(* CODESYS project Manutec_r2.project

Project tree, tasks and I/O mapping:
  Manutec : CODESYS SoftMotion Win V3, 3S - Smart Software Solutions GmbH, order no. 309021, version 3.5.9.20
    application Application
      libraries: SysSocket, * (System)
      task Manu_PlanningTask (cyclic, interval t#1000ms, priority 2) calls Manutech_PlanningPrg, Server
      task Task (cyclic, interval t#20ms, priority 1) calls RoboterSteuerung, qSoll
      task VISU_TASK (cyclic, interval 100 ms, priority 31) calls VisuElems.Visu_Prg
      axis group Manutech: TRAFO.Kin_ArticulatedRobot_6DOF, axes DriveA1, DriveA2, DriveA3, DriveA4, DriveA5, DriveA6
      program Manutech_PlanningPrg [ST]
      program RoboterSteuerung [FBD]
      global variables GVL
      visualisation Visualization
      visualisation VIS_Arm2
      data type CLIENT_ACCEPT
      data type SOCKET_LINGER
      TCP/
        function TcpReceiveData [ST]
        function TcpSendData [ST]
        function TcpServerOpenSocket [ST]
        function TcpServerWaitForConnect [ST]
        function block Tcp_Server [ST]
      program Server [FBD]
      program qSoll [ST]
    SoftMotion General Axis Pool
      DriveA1 : SM_Drive_Virtual, 3S - Smart Software Solutions GmbH, order no. 1805, version 4.0.0.0
          settings: wDriveID = 0; fSWMaxAcceleration = 100; fSWMaxDeceleration = 100; fSWMaxJerk = 1000; fSWLimitPositive = 360; fSWLimitNegative = 0; fSWLimitDeceleration = 0.0; fSWErrorMaxDistance = 0.0
      DriveA2 : SM_Drive_Virtual, 3S - Smart Software Solutions GmbH, order no. 1805, version 4.0.0.0
          settings: fSWMaxAcceleration = 100; fSWMaxDeceleration = 100; fSWMaxJerk = 1000; fSWLimitPositive = 90; fSWLimitNegative = -90
      DriveA3 : SM_Drive_Virtual, 3S - Smart Software Solutions GmbH, order no. 1805, version 4.0.0.0
          settings: wDriveID = 2; fSWLimitPositive = 180; fSWLimitNegative = -180; bSWLimitEnable = TRUE
      DriveA4 : SM_Drive_Virtual, 3S - Smart Software Solutions GmbH, order no. 1805, version 4.0.0.0
          settings: wDriveID = 3
      DriveA5 : SM_Drive_Virtual, 3S - Smart Software Solutions GmbH, order no. 1805, version 4.0.0.0
          settings: wDriveID = 4
      DriveA6 : SM_Drive_Virtual, 3S - Smart Software Solutions GmbH, order no. 1805, version 4.0.0.0
          settings: wDriveID = 5
  text list GlobalTextList
*)

// Manutec/Application/CLIENT_ACCEPT
TYPE  CLIENT_ACCEPT :
STRUCT
	Socket:DINT;       (* Socket Id des Client  *)
	IPAddress:STRING(20);	(* IP Adresse des Client *)
END_STRUCT
END_TYPE

// Manutec/Application/SOCKET_LINGER
TYPE  SOCKET_LINGER :
STRUCT
	l_onoff:WORD;
	l_linger:WORD;
END_STRUCT
END_TYPE

// Manutec/Application/GVL
VAR_GLOBAL CONSTANT
	PI: REAL := 3.141592654;
END_VAR
VAR_GLOBAL
	AxisMove: BOOL;
	PtpMOVE : BOOL;
	MoveLin: BOOL;
	Ziel : SMC_POS_REF;
	SOCKET_INVALID : DINT := -1;
	Port:INT:=2000;
	qAct:ARRAY[1..8] OF REAL;;
END_VAR

// Manutec/Application/Manutech_PlanningPrg
PROGRAM Manutech_PlanningPrg

;

END_PROGRAM

// Manutec/Application/Server
PROGRAM  Server
VAR
		Server: TCP_Server;
END_VAR

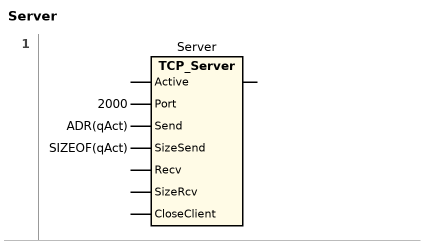
// NETWORK 1
Server(Port := 2000, Send := ADR(qAct), SizeSend := SIZEOF(qAct)); // TCP_Server

END_PROGRAM

// Manutec/Application/TCP/Tcp_Server
FUNCTION_BLOCK Tcp_Server
VAR_INPUT
	Active: BOOL;
	Port : INT;							(* zum Datenaustausch verwendeter Port *)
	Send : DWORD;					(* Sende Daten *)
	SizeSend : DINT;
	Recv : DWORD;					(* Empfangs Daten *)
	SizeRcv : DINT;
	CloseClient: BOOL;							(*Client schließen*)
END_VAR
VAR_OUTPUT

END_VAR
VAR
	Socket : DINT := -1;						(* Socket Id (wird von FUN "TcpServerOpenSocket" erzeugt) *)
	Client : CLIENT_ACCEPT := (Socket := -1);


END_VAR

IF Active THEN		(* Wenn Server aktiv dann ... *)
	IF Socket = -1 THEN		(* Wenn noch kein Server Socket geöffnet, dann ... *)
		Socket := TcpServerOpenSocket(Port, 10, 1000); (* ... Server Socket öffnen *)
		END_IF
	IF  Client.Socket = -1 THEN		(* Wenn noch kein Client verbuden, dann...   *)
		Client := TcpServerWaitForConnect(Socket, 4);	(*... warten auf Verbindung*)
	END_IF
	IF  Client.Socket <> -1 THEN	(* Wenn ein Client verbuden, dann...   *)
		TcpSendData(Client.Socket, Send, SizeSend, 1);		(* ... Daten senden *)
		TcpReceiveData(Client.Socket, Recv, SizeRcv, 5);	(* Daten empfangen *)
	END_IF
	IF CloseClient THEN		(* Wenn Client geschlossen werden soll, dann... *)
		CloseClient := FALSE;		(* ... Schließbefehl wieder auf FALSE setzen   *)
		SysSockClose(hSocket:=Client.Socket);	(* Client Socket schließen  *)
		Client.Socket := -1;		(* Client Socket wieder auf Startwert setzen *)
	END_IF
END_IF

END_FUNCTION_BLOCK

// Manutec/Application/TCP/TcpServerOpenSocket
FUNCTION TcpServerOpenSocket :  DINT
(*	Open a TCP server socket.
	Return:	Main Socket Id
*)
VAR_INPUT
	iPort:INT;						(* Port number *)
	diMaxConnections:DINT;		(* Max possible client connections of the server *)
	diMaxDataSize:DINT;			(* Max size of data to transmitt; if size = 0 default values are used *)
END_VAR
VAR
	diSocket:DINT;
	pResult:UDINT;  //Funktion überprüfen
	sa:SOCKADDRESS;
	bOptNoDelay:BOOL;
	lOptLinger:SOCKET_LINGER;
	
END_VAR

diSocket:=SysSockCreate(SOCKET_AF_INET, SOCKET_STREAM, 0, pResult);
IF diSocket <> SOCKET_INVALID THEN
(*
	IF diMaxDataSize <> 0 THEN
		SysSockSetOption(diSocket, SOCKET_SOL, SOCKET_SO_SNDBUF, ADR(diMaxDataSize), SIZEOF(diMaxDataSize));
		SysSockSetOption(diSocket, SOCKET_SOL, SOCKET_SO_RCVBUF, ADR(diMaxDataSize), SIZEOF(diMaxDataSize));
	END_IF
	lOptLinger.l_onoff:=0;
	lOptLinger.l_linger:=0;
	SysSockSetOption(diSocket,	SOCKET_SOL, SOCKET_SO_LINGER, ADR(lOptLinger), SIZEOF(lOptLinger));
	bOptNoDelay:=TRUE;
	SysSockSetOption(diSocket,	SOCKET_IPPROTO_TCP, SOCKET_TCP_NODELAY, ADR(bOptNoDelay), SIZEOF(bOptNoDelay));
*)

	sa.sin_family:=SOCKET_AF_INET;
	sa.sin_addr.ulAddr:=SOCKET_INADDR_ANY;
	sa.sin_port:=SysSockHtons(iPort);
	pResult:=SysSockBind(diSocket, ADR(sa), SIZEOF(sa));
	IF pResult >0 THEN
		diSocket:=SOCKET_INVALID;
	ELSE
		pResult:=SysSockListen(diSocket, diMaxConnections);
		IF pResult >0 THEN
			diSocket:=SOCKET_INVALID;
		END_IF
	END_IF
END_IF
TcpServerOpenSocket:=diSocket;

END_FUNCTION

// Manutec/Application/TCP/TcpServerWaitForConnect
FUNCTION TcpServerWaitForConnect : CLIENT_ACCEPT
(*	Wait for a TCP client to connect.
	ATTENTION:  Function is blocking, until a client tries to connect!
	Return:	diSocket : Socket Id for connection session
				stIPAddress : IP-Address of connected client
*)
VAR_INPUT
	diServerSocket:DINT;
	diTimeout : DINT;	(* Timeout in seconds *)
END_VAR
VAR
	sa:SOCKADDRESS;
	ia:INADDR;
	diSize:DINT;
	presult : UDINT;    //funktion überprüfen
	fdRead: SOCKET_FD_SET;
	fdWrite:SOCKET_FD_SET;
	fdExcept:SOCKET_FD_SET;
	tvTimeout:SOCKET_TIMEVAL;
END_VAR

tvTimeout.tv_sec := diTimeout ;
tvTimeout.tv_usec := 0;
fdRead.fd_count := 1;
fdRead.fd_array[0] := diServerSocket;
IF (SysSockSelect(SOCKET_FD_SETSIZE, ADR(fdRead), 0, 0, ADR(tvTimeout),pResult) > 0) THEN
	diSize:=SIZEOF(sa);
	TcpServerWaitForConnect.Socket:=SysSockAccept(diServerSocket, ADR(sa), ADR(diSize),pResult);
	ia.ulAddr:=DINT_TO_DWORD(sa.sin_addr.ulAddr);
	SysSockInetNtoa(ADR(ia), TcpServerWaitForConnect.IPAddress, SIZEOF(TcpServerWaitForConnect.IPAddress));
ELSE
	TcpServerWaitForConnect.Socket := -1;
END_IF

END_FUNCTION

// Manutec/Application/TCP/TcpSendData
FUNCTION TcpSendData :  DINT
(*	Send data via TCP socket.
	Return:	Number of bytes sent
*)
VAR_INPUT
	diSocket:DINT;		(* Socket Id *)
	pbyData:DWORD;		(* Address of data buffer *)
	diDataSize:DINT;		(* Size of data to send *)
	diTImeout : DINT;		(* Timeout in seconds *)
END_VAR
VAR
	fdWrite:SOCKET_FD_SET;
	tvTimeout:SOCKET_TIMEVAL;
	presult : UDINT;
	pdiReady : UDINT;
END_VAR

tvTimeout.tv_sec := diTimeout ;
tvTimeout.tv_usec := 0;
fdWrite.fd_count := 1;
fdWrite.fd_array[0] := diSocket;
//Funktion von SysSockSelect noch überprüfen, pdiReady sollte >0 sein (Anzahl der Sockets)
IF (SysSockSelect(SOCKET_FD_SETSIZE, 0, ADR(fdWrite), 0, ADR(tvTimeout),pdiReady) > 0) THEN
	TcpSendData:=SysSockSend(diSocket, pbyData, diDataSize, 0,pResult);
END_IF

END_FUNCTION

// Manutec/Application/TCP/TcpReceiveData
FUNCTION TcpReceiveData :  DINT
(*	Receive data from a tcp socket.
	Return:	Number of bytes received
*)
VAR_INPUT
	diSocket:DINT;		(* Socket Id *)
	pbyData:DWORD;		(* Address of data buffer *)
	diDataSize:DINT;		(* Size of data to send *)
	diTImeout : DINT;		(* Timeout in seconds *)
END_VAR
VAR
	fdRead:SOCKET_FD_SET;
	tvTimeout:SOCKET_TIMEVAL;
	presult : UDINT;
	pdiReady : UDINT;
END_VAR

tvTimeout.tv_sec := diTimeout ;
tvTimeout.tv_usec := 0;
fdRead.fd_count := 1;
fdRead.fd_array[0] := diSocket;
//Funktion von SysSockSelect noch überprüfen, pdiReady sollte >0 sein (Anzahl der Sockets)
IF (SysSockSelect(SOCKET_FD_SETSIZE, ADR(fdRead), 0, 0, ADR(tvTimeout),pdiReady) > 0) THEN
	TcpReceiveData:=SysSockRecv(diSocket, pbyData, diDataSize, 0,pdiReady);
END_IF

END_FUNCTION

// Manutec/Application/RoboterSteuerung
PROGRAM RoboterSteuerung
VAR
	MoveAxisDirect: MC_MoveDirectAbsolute;
	Roboter: MC_GroupEnable;
	E1, E2, E3, E4, E5, E6: MC_Power;
	Axes: MC_GroupReadActualPosition;
	TCP: MC_GroupReadActualPosition;
	MovePtp: MC_MoveDirectAbsolute;
	MoveLinear: MC_MoveLinearAbsolute;
END_VAR

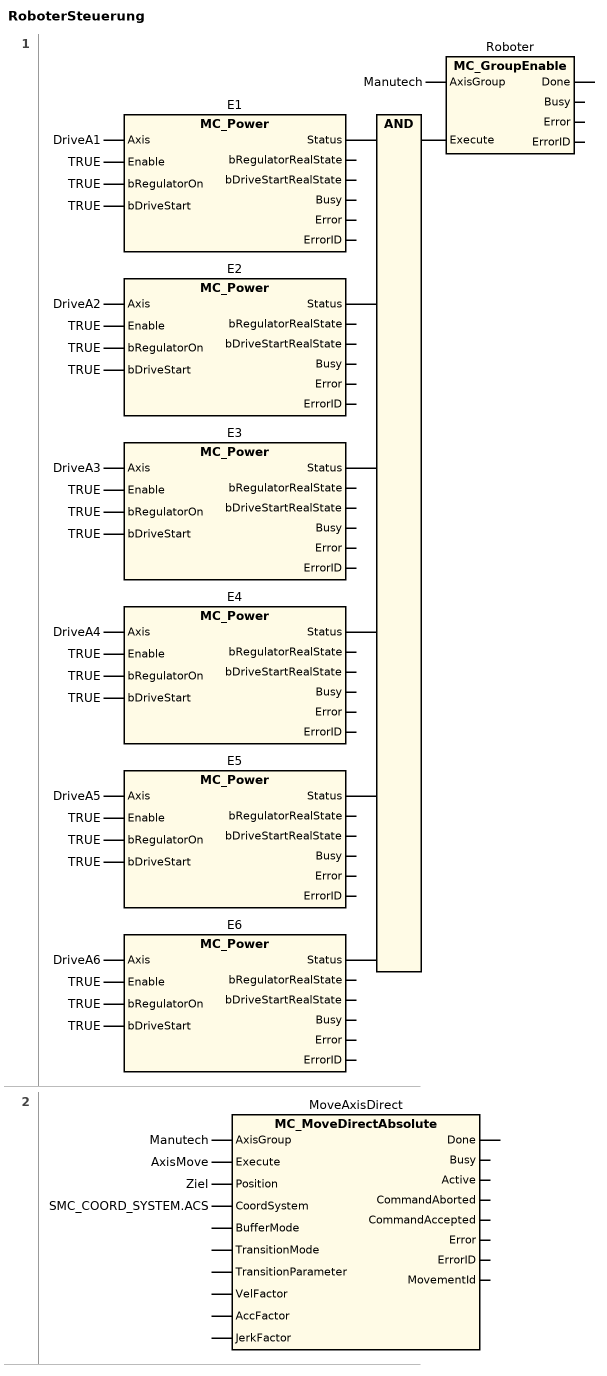
// NETWORK 1
E1(Axis := DriveA1, Enable := TRUE, bRegulatorOn := TRUE, bDriveStart := TRUE); // MC_Power
E2(Axis := DriveA2, Enable := TRUE, bRegulatorOn := TRUE, bDriveStart := TRUE); // MC_Power
E3(Axis := DriveA3, Enable := TRUE, bRegulatorOn := TRUE, bDriveStart := TRUE); // MC_Power
E4(Axis := DriveA4, Enable := TRUE, bRegulatorOn := TRUE, bDriveStart := TRUE); // MC_Power
E5(Axis := DriveA5, Enable := TRUE, bRegulatorOn := TRUE, bDriveStart := TRUE); // MC_Power
E6(Axis := DriveA6, Enable := TRUE, bRegulatorOn := TRUE, bDriveStart := TRUE); // MC_Power
Roboter(AxisGroup := Manutech, Execute := E1.Status AND E2.Status AND E3.Status AND E4.Status AND E5.Status AND E6.Status); // MC_GroupEnable

// NETWORK 2
MoveAxisDirect(
    AxisGroup := Manutech,
    Execute := AxisMove,
    Position := Ziel,
    CoordSystem := SMC_COORD_SYSTEM.ACS); // MC_MoveDirectAbsolute

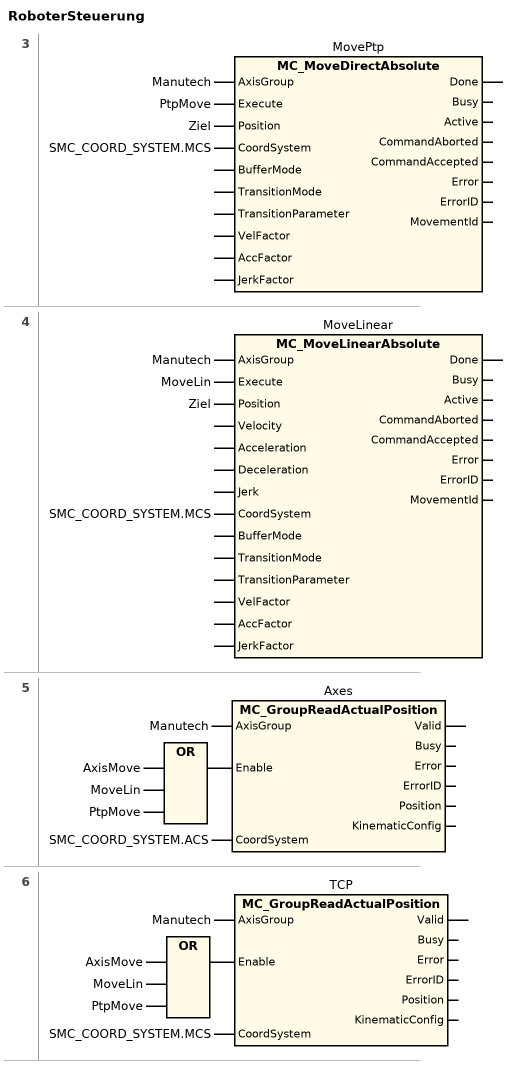
// NETWORK 3
MovePtp(AxisGroup := Manutech, Execute := PtpMove, Position := Ziel, CoordSystem := SMC_COORD_SYSTEM.MCS); // MC_MoveDirectAbsolute

// NETWORK 4
MoveLinear(AxisGroup := Manutech, Execute := MoveLin, Position := Ziel, CoordSystem := SMC_COORD_SYSTEM.MCS); // MC_MoveLinearAbsolute

// NETWORK 5
Axes(AxisGroup := Manutech, Enable := AxisMove OR MoveLin OR PtpMove, CoordSystem := SMC_COORD_SYSTEM.ACS); // MC_GroupReadActualPosition

// NETWORK 6
TCP(AxisGroup := Manutech, Enable := AxisMove OR MoveLin OR PtpMove, CoordSystem := SMC_COORD_SYSTEM.MCS); // MC_GroupReadActualPosition

END_PROGRAM

// Manutec/Application/qSoll
PROGRAM qSoll
VAR
	
END_VAR



qAct[1]:=LREAL_TO_REAL(RoboterSteuerung.Axes.Position.a.a0);
qAct[2]:=LREAL_TO_REAL(RoboterSteuerung.Axes.Position.a.a1);
qAct[3]:=LREAL_TO_REAL(RoboterSteuerung.Axes.Position.a.a2);
qAct[4]:=LREAL_TO_REAL(RoboterSteuerung.Axes.Position.a.a3);
qAct[5]:=LREAL_TO_REAL(RoboterSteuerung.Axes.Position.a.a4);
qAct[6]:=LREAL_TO_REAL(RoboterSteuerung.Axes.Position.a.a5);
qAct[7]:=0;
qAct[8]:=0;

END_PROGRAM

// Manutec/Application/Visualization
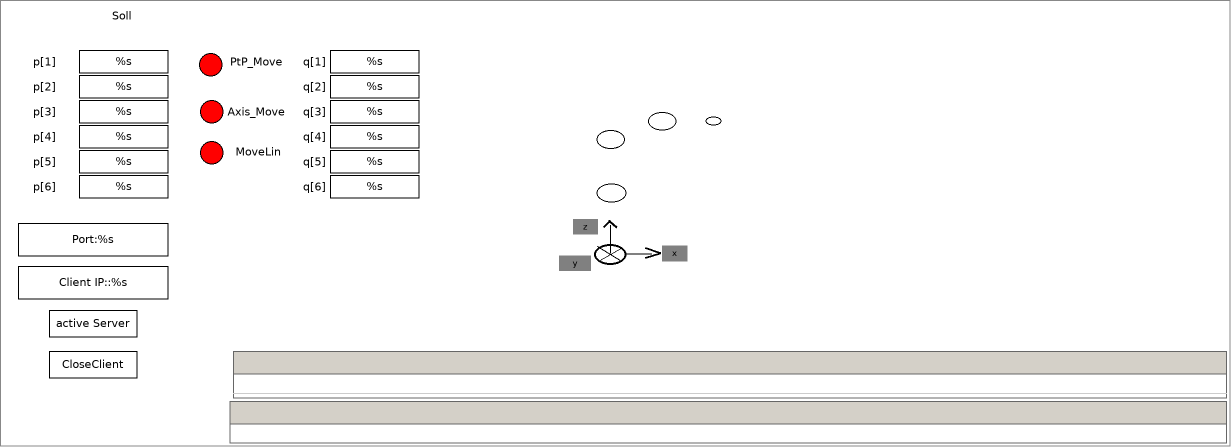
VISUALIZATION Visualization  // 1231x447
    Frame (219,19 1010x426)
        shows VIS_Arm2(qAct := RoboterSteuerung.Axes.Position.a, pAct := RoboterSteuerung.TCP.Position.c)
    Rectangle (220,50 73x24), "PtP_Move"
    Ellipse (199,53 23x23), colour toggle: PtpMove
        toggle PtpMove
    Rectangle (300,50 31x24), "q[1]"
    Rectangle (108,4 28x24), "Soll"
    Rectangle (300,75 31x24), "q[2]"
    Rectangle (30,50 31x24), "p[1]"
    Rectangle (30,75 30x24), "p[2]"
    Rectangle (330,50 89x23), "%s", text variable: Ziel.a.a0
        OnMouseDown: write the text variable via Edit
    Rectangle (330,75 89x23), "%s", text variable: Ziel.a.a1
        OnMouseDown: write the text variable via Edit
    Rectangle (79,50 89x23), "%s", text variable: Ziel.c.X
        OnMouseDown: write the text variable via Edit
    Rectangle (79,75 89x23), "%s", text variable: Ziel.c.Y
        OnMouseDown: write the text variable via Edit
    Rectangle (220,100 73x24), "Axis_Move"
    Ellipse (200,100 23x23), colour toggle: AxisMove
        toggle AxisMove
    Rectangle (79,100 89x23), "%s", text variable: Ziel.c.Z
        OnMouseDown: write the text variable via Edit
    Rectangle (30,100 29x24), "p[3]"
    Rectangle (30,125 29x24), "p[4]"
    Rectangle (30,150 29x24), "p[5]"
    Rectangle (30,175 29x24), "p[6]"
    Rectangle (79,125 89x23), "%s", text variable: Ziel.c.A
        OnMouseDown: write the text variable via Edit
    Rectangle (79,150 89x23), "%s", text variable: Ziel.c.B
        OnMouseDown: write the text variable via Edit
    Rectangle (79,175 89x23), "%s", text variable: Ziel.c.C
        OnMouseDown: write the text variable via Edit
    Rectangle (300,100 31x24), "q[3]"
    Rectangle (300,125 31x24), "q[4]"
    Rectangle (300,150 31x24), "q[5]"
    Rectangle (300,175 31x24), "q[6]"
    Rectangle (330,100 89x23), "%s", text variable: Ziel.a.a2
        OnMouseDown: write the text variable via Edit
    Rectangle (330,150 89x23), "%s", text variable: Ziel.a.a4
        OnMouseDown: write the text variable via Edit
    Rectangle (330,125 89x23), "%s", text variable: Ziel.a.a3
        OnMouseDown: write the text variable via Edit
    Rectangle (330,175 89x23), "%s", text variable: Ziel.a.a5
        OnMouseDown: write the text variable via Edit
    Ellipse (200,141 23x23), colour toggle: MoveLin
        toggle MoveLin
    Rectangle (224,140 69x24), "MoveLin"
    Rectangle (18,223 150x33), "Port:%s", text variable: Server.Server.Port
    Rectangle (18,266 150x33), "Client IP::%s", text variable: Server.Server.Client.IPAddress
    Rectangle (49,310 88x27), "active Server", colour toggle: Server.Server.Active
        toggle Server.Server.Active
    Rectangle (49,351 88x27), "CloseClient", colour toggle: Server.Server.CloseClient
        tap Server.Server.CloseClient
END_VISUALIZATION

// Manutec/Application/VIS_Arm2
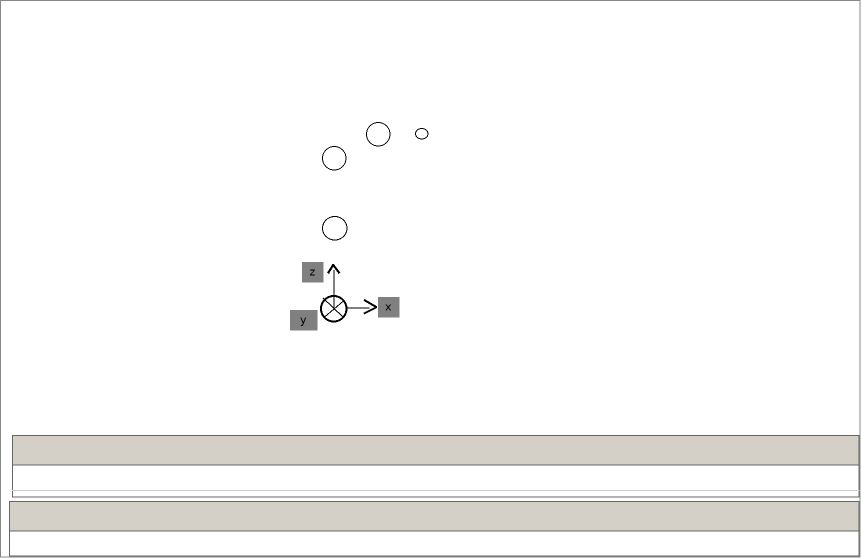
VISUALIZATION VIS_Arm2  // 861x558
VAR_IN_OUT(*	qAct:ARRAY[1..6] OF REAL;*)
	qAct:TRAFO.AXISPOS_REF;
	pAct:MC_COORD_REF;
END_VAR
    Table (9,501 850x55), data array: qAct
        p3854506369: qAct.a0
        p1892666644: qAct.a1
        p338671338: qAct.a2
        p2170511999: qAct.a3
        p3723444502: qAct.a4
        p1218418051: qAct.a5
    Table (12,435 847x62), data array: pAct
        p3854506369: pAct.X
        p1892666644: pAct.Y
        p338671338: pAct.Z
        p2170511999: pAct.A
        p3723444502: pAct.B
        p1218418051: pAct.C
    Polygon (24,225)
    Polygon (65,175)
        p2858320360: qAct.a1
    Polygon (76,225)
    Polygon (65,105)
        p3560616238: 70 *SIN(qAct.a1*PI/180)
        p2738717112: 70*(1- COS(qAct.a1*PI/180))
        p2858320360: (qAct.a2)
    Ellipse (322,216 25x24)
    Ellipse (322,146 24x24)
        p3560616238: 70 *SIN(qAct.a1*PI/180)
        p2738717112: 70*(1-COS(qAct.a1*PI/180))
        p2858320360: (qAct.a2)
    Polygon (65,105)
        p3560616238: 70 *SIN(qAct.a1*PI/180)
        p2738717112: 70*(1- COS(qAct.a1*PI/180))
        p2858320360: (qAct.a2)
    Ellipse (415,128 13x11)
        p3560616238: 70 *SIN(qAct.a1*PI/180) +30*(COS(qAct.a2*PI/180)-1)
        p2738717112: 70*(1- COS(qAct.a1*PI/180))+60*(SIN(qAct.a2*PI/180))
        p2858320360: (qAct.a4)
    Line (369,308) (335,308)
    Ellipse (320,295 27x27)
    Polyline (364,313) (376,307) (364,300)
    Polyline (328,273) (333,265) (339,273)
    Rectangle (378,297 21x20), "x"
    Rectangle (290,310 27x20), "y"
    Rectangle (302,262 21x20), "z"
    Line (343,301) (324,317)
    Line (343,317) (323,298)
    Polygon (65,105)
        p3560616238: 70 *SIN(qAct.a1*PI/180) +30*(COS(qAct.a2*PI/180)-1)
        p2738717112: 70*(1- COS(qAct.a1*PI/180))+60*(SIN(qAct.a2*PI/180))
        p2858320360: (qAct.a4)
    Line (334,307) (334,270)
    Ellipse (366,122 24x24)
        p3560616238: 70 *SIN(qAct.a1*PI/180)
        p2738717112: 70*(1-COS(qAct.a1*PI/180))
        p2858320360: (qAct.a2)
END_VISUALIZATION
